Yaskawa INFORM job: OK_R2_O49(180,90)AWOK.JBI

/JOB
//NAME OK_R2_O49(180,90)AWOK
///FOLDERNAME X4
//POS
///NPOS 112,112,112,7,0,0
///TOOL 0
///POSTYPE PULSE
///PULSE
C00000=57370,-49169,-35389,92398,112235,-2416
C00001=57338,-39846,-12309,87938,111954,-7208
C00002=61668,-40068,-12639,88811,108884,-7066
C00003=63399,-40053,-12708,89154,107656,-7009
C00004=65644,-43123,-14595,89423,106041,-7176
C00005=66050,-42449,-14221,89539,105759,-7114
C00006=65644,-43123,-14595,89423,106041,-7176
C00007=63399,-40053,-12708,89154,107656,-7009
C00008=65860,-35872,-10226,89816,105931,-6667
C00009=67308,-37830,-11473,89989,104891,-6764
C00010=65860,-35872,-10226,89816,105931,-6667
C00011=63399,-40053,-12708,89154,107656,-7009
C00012=61668,-40068,-12639,88811,108884,-7066
C00013=57338,-39846,-12309,87938,111954,-7208
C00014=57370,-49169,-35389,92398,112235,-2416
C00015=56766,-48274,-34752,92403,112675,-2380
C00016=56734,-38983,-11654,87839,112385,-7203
C00017=61035,-39257,-12018,88706,109335,-7062
C00018=61363,-41475,-13444,88660,109088,-7185
C00019=65079,-42508,-14107,89322,106443,-7178
C00020=65354,-42062,-13862,89401,106251,-7134
C00021=65079,-42508,-14107,89322,106443,-7178
C00022=62757,-39264,-12100,89046,108114,-7005
C00023=65205,-35368,-10154,89778,106406,-6571
C00024=66729,-37471,-11499,89953,105309,-6677
C00025=65205,-35368,-10154,89778,106406,-6571
C00026=62757,-39264,-12100,89046,108114,-7005
C00027=61035,-39257,-12018,88706,109335,-7062
C00028=56734,-38983,-11654,87839,112385,-7203
C00029=56766,-48274,-34752,92403,112675,-2380
C00030=56218,-47521,-34536,92505,113073,-2248
C00031=56187,-38348,-11498,87842,112791,-7100
C00032=59131,-40673,-13118,88322,110687,-7128
C00033=64463,-43713,-15068,89195,106879,-7202
C00034=65258,-42417,-14335,89420,106324,-7084
C00035=65041,-42755,-14501,89355,106475,-7122
C00036=62171,-38696,-11986,89025,108542,-6906
C00037=64564,-34510,-9127,89599,106856,-6674
C00038=65923,-36436,-10368,89757,105878,-6764
C00039=64564,-34510,-9127,89599,106856,-6674
C00040=62171,-38696,-11986,89025,108542,-6906
C00041=60460,-38670,-11893,88691,109758,-6961
C00042=56187,-38348,-11498,87842,112791,-7100
C00043=58012,-44746,-32893,92770,111760,-2043
C00044=166129,-61778,-24330,-90630,98825,8752
C00045=158947,-59821,-23656,-92312,93807,8452
C00046=157694,-61727,-24710,-92552,92933,8610
C00047=156488,-58840,-23278,-92861,92081,8335
C00048=157694,-61727,-24710,-92552,92933,8610
C00049=160818,-58525,-23006,-91940,95118,8328
C00050=158550,-54892,-21231,-92501,93522,7967
C00051=157594,-55549,-21576,-92682,92849,8027
C00052=159188,-54439,-20992,-92380,93971,7927
C00053=166129,-61778,-24330,-90630,98825,8752
C00054=167320,-61671,-24024,-90329,99652,8826
C00055=160101,-59851,-23419,-92043,94615,8527
C00056=157289,-61712,-24386,-92627,92650,8699
C00057=156480,-59783,-23436,-92835,92081,8513
C00058=156648,-62103,-24576,-92764,92203,8740
C00059=161059,-59179,-23083,-91852,95286,8462
C00060=158397,-53862,-21182,-92580,93409,7736
C00061=157302,-54629,-21597,-92783,92637,7805
C00062=159439,-53107,-20779,-92391,94146,7669
C00063=167320,-61671,-24024,-90329,99652,8826
C00064=168043,-60879,-23856,-90231,100166,8690
C00065=160879,-59137,-23279,-91909,95160,8396
C00066=157512,-61415,-24459,-92595,92804,8607
C00067=156739,-59612,-23633,-92794,92258,8414
C00068=157512,-61415,-24459,-92595,92804,8607
C00069=162331,-58072,-22741,-91629,96179,8297
C00070=160316,-53391,-20502,-92182,94764,7816
C00071=158516,-54703,-21211,-92514,93496,7928
C00072=160111,-53544,-20583,-92219,94619,7829
C00073=168043,-60879,-23856,-90231,100166,8690
C00074=70363,-72912,-29776,103135,36074,80294
C00075=72045,-74207,-30319,104357,35005,79859
C00076=72656,-65874,-14855,122721,41176,74315
C00077=71246,-73594,-30065,103766,35512,80070
C00078=71620,-76170,-31054,104938,35409,79478
C00079=73197,-57217,-1310,126820,42940,71941
C00080=73676,-56716,-1016,127117,42645,71869
C00081=74247,-46779,14189,131192,44872,69470
C00082=74488,-59138,-6611,125662,40993,72927
C00083=74963,-49474,8604,130071,43270,70357
C00084=75571,-57025,-4682,126589,40456,72598
C00085=75843,-46558,11852,131203,43136,69869
C00086=76543,-55367,-3431,127266,39884,72395
C00087=76901,-45590,12066,131763,42396,69788
C00088=77467,-63691,-18308,122675,36762,75194
C00089=77943,-54955,-4053,127787,38793,72371
C00090=78454,-64206,-20641,121996,35600,75720
C00091=78974,-55395,-6053,127565,37664,72694
C00092=57457,-68163,-11759,115838,51418,75388
C00093=67053,-69065,-28106,99490,40183,-15728
C00094=67428,-69282,-26772,100738,40056,-16409
C00095=67260,-59795,-12797,115520,44608,-22426
C00096=65920,-70446,-28647,99537,41009,-15920
C00097=68407,-70268,-28636,100327,39293,-16023
C00098=67784,-51665,588,119520,46005,-24885
C00099=68275,-59835,-14059,115360,43685,-22125
C00100=68716,-51078,50,119546,45176,-24682
C00101=69246,-59613,-14754,115378,42870,-21962
C00102=69751,-50486,-158,119823,44377,-24633
C00103=70142,-59710,-16598,114777,41891,-21440
C00104=70635,-50550,-1374,119731,43536,-24387
C00105=71343,-49966,-1072,120083,43069,-24462
C00106=71667,-39030,16614,125050,45509,-27517
C00107=72039,-64081,-28414,110138,38936,-18430
C00108=72373,-56232,-14851,115286,40209,-21389
C00109=72508,-46257,2157,120937,42429,-24750
C00110=72834,-35448,19521,125853,44865,-27742
C00111=71161,-41775,15932,125497,46306,-27939
BC00000=398158,464340,70906
BC00001=398158,464340,70906
BC00002=398158,464340,70906
BC00003=398158,464340,70906
BC00004=398158,464340,70906
BC00005=398158,464340,70906
BC00006=398158,464340,70906
BC00007=398158,464340,70906
BC00008=398158,464340,70906
BC00009=398158,464340,70906
BC00010=398158,464340,70906
BC00011=398158,464340,70906
BC00012=398158,464340,70906
BC00013=398158,464340,70906
BC00014=398158,464340,70906
BC00015=398158,469239,420555
BC00016=398158,469239,420555
BC00017=398158,469239,420555
BC00018=398158,469239,420555
BC00019=398158,469239,420555
BC00020=398158,469239,420555
BC00021=398158,469239,420555
BC00022=398158,469239,420555
BC00023=398158,469239,420555
BC00024=398158,469239,420555
BC00025=398158,469239,420555
BC00026=398158,469239,420555
BC00027=398158,469239,420555
BC00028=398158,469239,420555
BC00029=398158,469239,420555
BC00030=398158,473961,751886
BC00031=398158,473961,751886
BC00032=398158,473961,751886
BC00033=398158,473961,751886
BC00034=398158,473961,751886
BC00035=398158,473961,751886
BC00036=398158,473961,751886
BC00037=398158,473961,751886
BC00038=398158,473961,751886
BC00039=398158,473961,751886
BC00040=398158,473961,751886
BC00041=398158,473961,751886
BC00042=398158,473961,751886
BC00043=398158,500538,751886
BC00044=1592,466255,63183
BC00045=1592,466255,63183
BC00046=1592,466255,63183
BC00047=1592,466255,63183
BC00048=1592,466255,63183
BC00049=1592,466255,63183
BC00050=1592,466255,63183
BC00051=1592,466255,63183
BC00052=1592,466255,63183
BC00053=1592,466255,63183
BC00054=1592,470033,395208
BC00055=1592,470033,395208
BC00056=1592,470033,395208
BC00057=1592,470033,395208
BC00058=1592,470033,395208
BC00059=1592,470033,395208
BC00060=1592,470033,395208
BC00061=1592,470033,395208
BC00062=1592,470033,395208
BC00063=1592,470033,395208
BC00064=1592,475695,759756
BC00065=1592,475695,759756
BC00066=1592,475695,759756
BC00067=1592,475695,759756
BC00068=1592,475695,759756
BC00069=1592,475695,759756
BC00070=1592,475695,759756
BC00071=1592,475695,759756
BC00072=1592,475695,759756
BC00073=1592,475695,759756
BC00074=1592,520429,870775
BC00075=1592,513222,869664
BC00076=1592,510340,869219
BC00077=1592,510340,869219
BC00078=1592,510340,869219
BC00079=1592,510340,869219
BC00080=1592,510340,794493
BC00081=1592,510340,794493
BC00082=1592,510340,652638
BC00083=1592,510340,652638
BC00084=1592,510340,530516
BC00085=1592,510340,530516
BC00086=1592,510340,409272
BC00087=1592,510340,409272
BC00088=1592,510340,241491
BC00089=1592,510340,241491
BC00090=1592,510340,105222
BC00091=1592,510340,105222
BC00092=1592,510340,105222
BC00093=308885,519368,873321
BC00094=311437,512513,872276
BC00095=311394,512565,872225
BC00096=312650,509257,871780
BC00097=312650,509257,871780
BC00098=311394,512565,872225
BC00099=311393,512558,750033
BC00100=311393,512558,750033
BC00101=311393,512558,629738
BC00102=311393,512558,629738
BC00103=311393,512558,498749
BC00104=311393,512558,498749
BC00105=311393,512558,426533
BC00106=311393,512558,426533
BC00107=311393,512558,186965
BC00108=311393,512558,186965
BC00109=311393,512558,186965
BC00110=311393,512558,186965
BC00111=311393,512558,186965
EC00000=-1596313,-740307
EC00001=-1596313,-740307
EC00002=-1596313,-740307
EC00003=-1596313,-740307
EC00004=-1596313,-740307
EC00005=-1596313,-740307
EC00006=-1596313,-740307
EC00007=-1596313,-740307
EC00008=-1596313,-740307
EC00009=-1596313,-740307
EC00010=-1596313,-740307
EC00011=-1596313,-740307
EC00012=-1596313,-740307
EC00013=-1596313,-740307
EC00014=-1596313,-740307
EC00015=-1596313,-740307
EC00016=-1596313,-740307
EC00017=-1596313,-740307
EC00018=-1596313,-740307
EC00019=-1596313,-740307
EC00020=-1596313,-740307
EC00021=-1596313,-740307
EC00022=-1596313,-740307
EC00023=-1596313,-740307
EC00024=-1596313,-740307
EC00025=-1596313,-740307
EC00026=-1596313,-740307
EC00027=-1596313,-740307
EC00028=-1596313,-740307
EC00029=-1596313,-740307
EC00030=-1596313,-740307
EC00031=-1596313,-740307
EC00032=-1596313,-740307
EC00033=-1596313,-740307
EC00034=-1596313,-740307
EC00035=-1596313,-740307
EC00036=-1596313,-740307
EC00037=-1596313,-740307
EC00038=-1596313,-740307
EC00039=-1596313,-740307
EC00040=-1596313,-740307
EC00041=-1596313,-740307
EC00042=-1596313,-740307
EC00043=-1596313,-740307
EC00044=-1596313,-740307
EC00045=-1596313,-740307
EC00046=-1596313,-740307
EC00047=-1596313,-740307
EC00048=-1596313,-740307
EC00049=-1596313,-740307
EC00050=-1596313,-740307
EC00051=-1596313,-740307
EC00052=-1596313,-740307
EC00053=-1596313,-740307
EC00054=-1596313,-740307
EC00055=-1596313,-740307
EC00056=-1596313,-740307
EC00057=-1596313,-740307
EC00058=-1596313,-740307
EC00059=-1596313,-740307
EC00060=-1596313,-740307
EC00061=-1596313,-740307
EC00062=-1596313,-740307
EC00063=-1596313,-740307
EC00064=-1596313,-740307
EC00065=-1596313,-740307
EC00066=-1596313,-740307
EC00067=-1596313,-740307
EC00068=-1596313,-740307
EC00069=-1596313,-740307
EC00070=-1596313,-740307
EC00071=-1596313,-740307
EC00072=-1596313,-740307
EC00073=-1596313,-740307
EC00074=-1596313,-740307
EC00075=-1596313,-740307
EC00076=-1596313,-740307
EC00077=-1596313,-740307
EC00078=-1596313,-740307
EC00079=-1596313,-740307
EC00080=-1596313,-740307
EC00081=-1596313,-740307
EC00082=-1596313,-740307
EC00083=-1596313,-740307
EC00084=-1596313,-740307
EC00085=-1596313,-740307
EC00086=-1596313,-740307
EC00087=-1596313,-740307
EC00088=-1596313,-740307
EC00089=-1596313,-740307
EC00090=-1596313,-740307
EC00091=-1596313,-740307
EC00092=-1596313,-740307
EC00093=-1596313,-740307
EC00094=-1596313,-740307
EC00095=-1596313,-740307
EC00096=-1596313,-740307
EC00097=-1596313,-740307
EC00098=-1596313,-740307
EC00099=-1596313,-740307
EC00100=-1596313,-740307
EC00101=-1596313,-740307
EC00102=-1596313,-740307
EC00103=-1596313,-740307
EC00104=-1596313,-740307
EC00105=-1596313,-740307
EC00106=-1596313,-740307
EC00107=-1596313,-740307
EC00108=-1596313,-740307
EC00109=-1596313,-740307
EC00110=-1596313,-740307
EC00111=-1596313,-740307
///POSTYPE BASE
///RECTAN
///RCONF 0,0,0,0,1,0,0,0,0,0,0,0,0,0,0,0,0,0,0,0,0,0,0,0
P00006=2.006,1.622,-0.565,0.0000,0.0000,0.0000
P00021=0.073,2.058,-0.109,0.0000,0.0000,0.0000
P00022=2.006,1.622,-0.565,0.0000,0.0000,0.0000
///RCONF 0,0,0,0,0,0,0,0,0,0,0,0,0,0,0,0,0,0,0,0,0,0,0,0
P00023=-2.957,-4.083,2.762,0.0000,0.0000,0.0000
P00031=-0.170,0.039,-0.647,0.0000,0.0000,0.0000
P00032=-0.423,0.157,3.222,0.0000,0.0000,0.0000
P00033=0.854,-1.099,3.047,0.0000,0.0000,0.0000
//INST
///DATE 2024/11/20 10:04
///ATTR SC,RW
///GROUP1 RB1,BS1
///GROUP2 ST1
NOP
'OK_r2_O49(180,90)
'Path S1126
SFTOF3D
MOVJ C00000 BC00000 VJ=100.00  +MOVJ EC00000 VJ=100.00
MOVJ C00001 BC00001 VJ=100.00  +MOVJ EC00001 VJ=100.00
MOVL C00002 BC00002 V=400.0  +MOVJ EC00002 VJ=100.00
SMOVL C00003 BC00003 V=100.0  +MOVJ EC00003
SMOVL C00004 BC00004 V=100.0  +MOVJ EC00004
SREFP 3 C00005 BC00005  +REFP EC00005
CALL JOB:SEARCH-R1-S13D
SET P031 P006
SFTON3D P031
SMOVL C00006 BC00006 V=100.0  +MOVJ EC00006
SMOVL C00007 BC00007 V=100.0  +MOVJ EC00007
SMOVL C00008 BC00008 V=100.0  +MOVJ EC00008
SREFP 3 C00009 BC00009  +REFP EC00009
CALL JOB:SEARCH-R1-S13D
SET P031 P006
SFTON3D P031
SMOVL C00010 BC00010 V=100.0  +MOVJ EC00010
SMOVL C00011 BC00011 V=100.0  +MOVJ EC00011
MOVL C00012 BC00012 V=400.0  +MOVJ EC00012 VJ=100.00
MOVL C00013 BC00013 V=1000.0  +MOVJ EC00013 VJ=100.00
MOVL C00014 BC00014 V=1000.0  +MOVJ EC00014 VJ=100.00
'Path S1127
SFTOF3D
MOVJ C00015 BC00015 VJ=100.00  +MOVJ EC00015 VJ=100.00
MOVJ C00016 BC00016 VJ=100.00  +MOVJ EC00016 VJ=100.00
MOVL C00017 BC00017 V=400.0  +MOVJ EC00017 VJ=100.00
SMOVL C00018 BC00018 V=100.0  +MOVJ EC00018
SMOVL C00019 BC00019 V=100.0  +MOVJ EC00019
SREFP 3 C00020 BC00020  +REFP EC00020
CALL JOB:SEARCH-R1-S13D
SET P032 P006
SFTON3D P032
SMOVL C00021 BC00021 V=100.0  +MOVJ EC00021
SMOVL C00022 BC00022 V=100.0  +MOVJ EC00022
SMOVL C00023 BC00023 V=100.0  +MOVJ EC00023
SREFP 3 C00024 BC00024  +REFP EC00024
CALL JOB:SEARCH-R1-S13D
SET P032 P006
SFTON3D P032
SMOVL C00025 BC00025 V=100.0  +MOVJ EC00025
SMOVL C00026 BC00026 V=100.0  +MOVJ EC00026
MOVL C00027 BC00027 V=400.0  +MOVJ EC00027 VJ=100.00
MOVL C00028 BC00028 V=1000.0  +MOVJ EC00028 VJ=100.00
MOVL C00029 BC00029 V=1000.0  +MOVJ EC00029 VJ=100.00
'Path S1128
SFTOF3D
MOVJ C00030 BC00030 VJ=100.00  +MOVJ EC00030 VJ=100.00
MOVJ C00031 BC00031 VJ=100.00  +MOVJ EC00031 VJ=100.00
MOVL C00032 BC00032 V=400.0  +MOVJ EC00032 VJ=100.00
SMOVL C00033 BC00033 V=100.0  +MOVJ EC00033
SREFP 3 C00034 BC00034  +REFP EC00034
CALL JOB:SEARCH-R1-S13D
SET P033 P006
SFTON3D P033
SMOVL C00035 BC00035 V=100.0  +MOVJ EC00035
SMOVL C00036 BC00036 V=100.0  +MOVJ EC00036
SMOVL C00037 BC00037 V=100.0  +MOVJ EC00037
SREFP 3 C00038 BC00038  +REFP EC00038
CALL JOB:SEARCH-R1-S13D
SET P033 P006
SFTON3D P033
SMOVL C00039 BC00039 V=100.0  +MOVJ EC00039
SMOVL C00040 BC00040 V=100.0  +MOVJ EC00040
MOVL C00041 BC00041 V=400.0  +MOVJ EC00041 VJ=100.00
MOVL C00042 BC00042 V=1000.0  +MOVJ EC00042 VJ=100.00
MOVL C00043 BC00043 V=1000.0  +MOVJ EC00043 VJ=100.00
'Path S1536
'DRUGA STRONA
'DRUGA STRONA
'DRUGA STRONA
SFTOF3D
MOVJ C00044 BC00044 VJ=100.00  +MOVJ EC00044 VJ=100.00
SMOVL C00045 BC00045 V=250.0  +MOVJ EC00045
SMOVL C00046 BC00046 V=100.0  +MOVJ EC00046
SREFP 3 C00047 BC00047  +REFP EC00047
CALL JOB:SEARCH-R1-S13D
SET P023 P006
SFTON3D P023
SMOVL C00048 BC00048 V=100.0  +MOVJ EC00048
SMOVL C00049 BC00049 V=100.0  +MOVJ EC00049
SMOVL C00050 BC00050 V=100.0  +MOVJ EC00050
SREFP 3 C00051 BC00051  +REFP EC00051
CALL JOB:SEARCH-R1-S13D
SET P023 P006
SFTON3D P023
SMOVL C00052 BC00052 V=100.0  +MOVJ EC00052
MOVL C00053 BC00053 V=1000.0  +MOVJ EC00053 VJ=100.00
'Path S1537
SFTOF3D
MOVJ C00054 BC00054 VJ=100.00  +MOVJ EC00054 VJ=100.00
SMOVL C00055 BC00055 V=250.0  +MOVJ EC00055
SMOVL C00056 BC00056 V=100.0  +MOVJ EC00056
SREFP 3 C00057 BC00057  +REFP EC00057
CALL JOB:SEARCH-R1-S13D
SET P022 P006
SFTON3D P022
SMOVL C00058 BC00058 V=100.0  +MOVJ EC00058
SMOVL C00059 BC00059 V=166.7  +MOVJ EC00059
SMOVL C00060 BC00060 V=100.0  +MOVJ EC00060
SREFP 3 C00061 BC00061  +REFP EC00061
CALL JOB:SEARCH-R1-S13D
SET P022 P006
SFTON3D P022
SMOVL C00062 BC00062 V=100.0  +MOVJ EC00062
MOVL C00063 BC00063 V=1000.0  +MOVJ EC00063 VJ=100.00
'Path S1538
SFTOF3D
MOVJ C00064 BC00064 VJ=100.00  +MOVJ EC00064 VJ=100.00
SMOVL C00065 BC00065 V=333.3  +MOVJ EC00065
SMOVL C00066 BC00066 V=100.0  +MOVJ EC00066
SREFP 3 C00067 BC00067  +REFP EC00067
CALL JOB:SEARCH-R1-S13D
SET P021 P006
SFTON3D P021
SMOVL C00068 BC00068 V=100.0  +MOVJ EC00068
SMOVL C00069 BC00069 V=166.7  +MOVJ EC00069
SMOVL C00070 BC00070 V=100.0  +MOVJ EC00070
SREFP 3 C00071 BC00071  +REFP EC00071
CALL JOB:SEARCH-R1-S13D
SET P021 P006
SFTON3D P021
SMOVL C00072 BC00072 V=100.0  +MOVJ EC00072
MOVL C00073 BC00073 V=1000.0  +MOVJ EC00073 VJ=100.00
'Path W1539
SFTOF3D
SFTON3D P021
MOVJ C00074 BC00074 VJ=100.00  +MOVJ EC00074 VJ=100.00
SMOVL C00075 BC00075 V=166.7  +MOVJ EC00075
SMOVL C00076 BC00076 V=133.3 PL=0  +MOVJ EC00076
SREFP 1 C00077 BC00077  +REFP EC00077
SREFP 2 C00078 BC00078  +REFP EC00078
MACRO1 MJ#(0) ARGF6
ARCON
SFTON3D P021
SMOVL C00079 BC00079 V=10.0  +MOVJ EC00079
ARCOF
SMOVL C00080 BC00080 V=500.0  +MOVJ EC00080
ARCON
SMOVL C00081 BC00081 V=10.0  +MOVJ EC00081
ARCOF
SFTON3D P022
SMOVL C00082 BC00082 V=500.0  +MOVJ EC00082
ARCON
SMOVL C00083 BC00083 V=10.0  +MOVJ EC00083
ARCOF
SMOVL C00084 BC00084 V=500.0  +MOVJ EC00084
ARCON
SMOVL C00085 BC00085 V=10.0  +MOVJ EC00085
ARCOF
SMOVL C00086 BC00086 V=500.0  +MOVJ EC00086
ARCON
SMOVL C00087 BC00087 V=10.0  +MOVJ EC00087
ARCOF
SFTON3D P023
SMOVL C00088 BC00088 V=500.0  +MOVJ EC00088
ARCON
SMOVL C00089 BC00089 V=10.0  +MOVJ EC00089
ARCOF
SMOVL C00090 BC00090 V=500.0  +MOVJ EC00090
ARCON
SMOVL C00091 BC00091 V=10.0  +MOVJ EC00091
ARCOF
SFTOF3D
MOVJ C00092 BC00092 VJ=100.00  +MOVJ EC00092 VJ=100.00
SFTOF3D
'Path W343
SFTOF3D
MOVJ C00093 BC00093 VJ=100.00  +MOVJ EC00093 VJ=100.00
SMOVL C00094 BC00094 V=400.0  +MOVJ EC00094
SFTON3D P033
SMOVL C00095 BC00095 V=133.3 PL=0  +MOVJ EC00095
SREFP 1 C00096 BC00096  +REFP EC00096
SREFP 2 C00097 BC00097  +REFP EC00097
MACRO1 MJ#(0) ARGF6
ARCON
SMOVL C00098 BC00098 V=10.0  +MOVJ EC00098
ARCOF
SMOVL C00099 BC00099 V=166.7  +MOVJ EC00099
ARCON
SMOVL C00100 BC00100 V=10.0  +MOVJ EC00100
ARCOF
SFTON3D P032
SMOVL C00101 BC00101 V=500.0  +MOVJ EC00101
ARCON
SMOVL C00102 BC00102 V=10.0  +MOVJ EC00102
ARCOF
SMOVL C00103 BC00103 V=500.0  +MOVJ EC00103
ARCON
SMOVL C00104 BC00104 V=10.0  +MOVJ EC00104
ARCOF
SFTON3D P031
SMOVL C00105 BC00105 V=500.0  +MOVJ EC00105
ARCON
SMOVL C00106 BC00106 V=10.0  +MOVJ EC00106
ARCOF
SFTON3D P031
SMOVL C00107 BC00107 V=500.0  +MOVJ EC00107
ARCON
SMOVL C00108 BC00108 V=10.0  +MOVJ EC00108
ARCOF
SMOVL C00109 BC00109 V=500.0  +MOVJ EC00109
ARCON
SMOVL C00110 BC00110 V=10.0  +MOVJ EC00110
ARCOF
SMOVL C00111 BC00111 V=1000.0  +MOVJ EC00111
SFTOF3D
END
